FUNCTION_BLOCK Sensor_MDL_RSP_PARSE
  (* Version 1.0, 2005-11-18, Goran Cengic, Chalmers *)
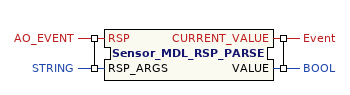
  EVENT_INPUT
    RSP : AO_EVENT WITH RSP_ARGS;
  END_EVENT
  EVENT_OUTPUT
    CURRENT_VALUE WITH VALUE;
  END_EVENT
  VAR_INPUT
    RSP_ARGS : STRING;
  END_VAR
  VAR_OUTPUT
    VALUE : BOOL;
  END_VAR
  VAR
    cmdArgs : STRING;
    cmd : INT;
  END_VAR
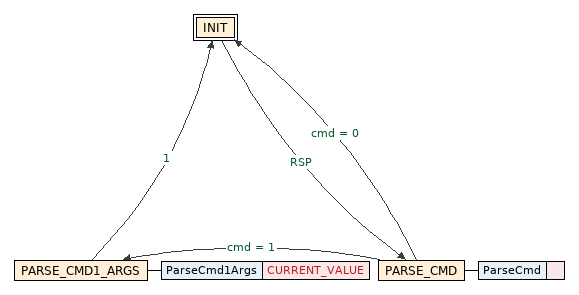
  EC_STATES
    INIT;
    PARSE_CMD : ParseCmd;
    PARSE_CMD1_ARGS : ParseCmd1Args -> CURRENT_VALUE;
  END_STATES
  EC_TRANSITIONS
    INIT TO PARSE_CMD := RSP;
    PARSE_CMD TO PARSE_CMD1_ARGS := cmd = 1;
    PARSE_CMD TO INIT := cmd = 0;
    PARSE_CMD1_ARGS TO INIT := 1;
  END_TRANSITIONS
  ALGORITHM ParseCmd IN Java:
	      cmd = RSP_ARGS.substring(0,RSP_ARGS.indexOf(' '));
	      if (cmd.toLowerCase().equals("current_value"))
		  {
		    cmd = 1;
			cmdArgs = RSP_ARGS.substring(RSP_ARGS.indexOf('	') + 1);
		  }
		  else
		  {
		    System.out.println("Sensor_MDL_RSP_PARSE: ParseCmd algorithm: Unknown command received on RSP_ARGS data input!");
		    cmd = 0;
		  }
  END_ALGORITHM
  ALGORITHM ParseCmd1Args IN Java:
	    VALUE = (new Boolean(cmdArgs)).booleanValue();
  END_ALGORITHM
END_FUNCTION_BLOCK
